INTERFACE I_CYLINDER_DA_TESTDEV2_4 EXTENDS I_CYLINDER_DA_GENERAL

METHOD M_OpenLockValves : BOOL
VAR_INPUT
  bOpenChA:        BOOL;
  bOpenChB:        BOOL;
END_VAR
END_METHOD

METHOD M_SetMaxPos : BOOL
VAR_INPUT
END_VAR
END_METHOD

METHOD M_SetZeroPos : BOOL
VAR_INPUT
END_VAR
END_METHOD

METHOD M_StopAndLock : BOOL
VAR_INPUT
END_VAR
END_METHOD

METHOD M_ToSetPos : BOOL
VAR_INPUT
  lrToSetPos:                 LREAL;
  /// Just need for prop valve
  eSpeedType:               E_SPEED_TYPE;
  rSpeed:                   REAL; 
END_VAR
END_METHOD

PROPERTY P_ActiveDirection : STRING
GET
END_GET
END_PROPERTY

PROPERTY P_DoubleActing : BOOL
GET
END_GET
END_PROPERTY

PROPERTY P_MaxPosVal : LREAL
GET
END_GET
END_PROPERTY

PROPERTY P_MinPosVal : LREAL
GET
END_GET
END_PROPERTY

PROPERTY P_Position : LREAL
GET
END_GET
END_PROPERTY

PROPERTY P_PositionAbs : LREAL
GET
END_GET
END_PROPERTY

PROPERTY P_PressureChA : REAL
GET
END_GET
END_PROPERTY

PROPERTY P_PressureChB : REAL
GET
END_GET
END_PROPERTY

PROPERTY P_SpeedInMmPerSecond : REAL
GET
END_GET
END_PROPERTY

PROPERTY P_SpeedInPercent : LREAL
GET
END_GET
END_PROPERTY

PROPERTY P_StrokeLength : REAL
GET
END_GET
END_PROPERTY

PROPERTY P_StrokeLengthInitialized : BOOL
GET
END_GET
SET
END_SET
END_PROPERTY

END_INTERFACE

(* stored: Version 1.1.0.1, ProductVersion 3.1.4024.12
   Itf I_CYLINDER_DA_TESTDEV2_4: Id {f16afa1c-8799-4f08-84e4-e0140353dd92}
   Method M_OpenLockValves: Id {2ca67dfe-0591-43a4-916c-384fb6af2657}
   Method M_SetMaxPos: Id {cea0ae47-e9bb-4f2e-bf7a-25e90d2d2955}
   Method M_SetZeroPos: Id {1ff466f2-f842-4159-9085-0bb5641ce510}
   Method M_StopAndLock: Id {74dc6512-611b-4bfe-84ef-8556535a1373}
   Method M_ToSetPos: Id {eded9da4-c374-40ff-b3c6-8b8ba669878d}
   Property P_ActiveDirection: Id {6203e25d-1d2e-4831-828b-3dd9d8c75aa4}
   Get Get: Id {7394b632-ea0c-48d3-9309-60833df95117}
   Property P_DoubleActing: Id {0b663a7c-7295-406b-b3e0-b046aa79acea}
   Get Get: Id {0442e461-205b-437a-97a8-3262d3e89e69}
   Property P_MaxPosVal: Id {75a29253-6f02-46db-8689-66b7709c9063}
   Get Get: Id {6d0277d3-aec1-4872-bee2-316417e4554c}
   Property P_MinPosVal: Id {3cce7030-0547-4c39-b29b-8a63b3db8061}
   Get Get: Id {818e9e8a-8ae0-49f1-8183-fb4253be33f4}
   Property P_Position: Id {aaf5d39b-950b-4fb4-9969-98f49b20be8b}
   Get Get: Id {bc82b54e-7ae4-4eab-8dd7-d6d38816469b}
   Property P_PositionAbs: Id {f5abc2d3-dc80-4dfb-9117-b9d4052ca3d4}
   Get Get: Id {22655590-92c2-4505-b7f6-7ba414aa1e6f}
   Property P_PressureChA: Id {2242dd50-d555-4854-9001-94346a7ea495}
   Get Get: Id {d7db13fa-f335-4081-9451-916fb814abc8}
   Property P_PressureChB: Id {07153e8d-795a-4709-a869-eb2aab084c16}
   Get Get: Id {b46329d2-2879-4ff8-8746-84792769ab21}
   Property P_SpeedInMmPerSecond: Id {301360ce-5962-4404-8936-dc0bc0f21f8a}
   Get Get: Id {9aeeef22-6037-4fbc-a70b-fc7a5fde3f85}
   Property P_SpeedInPercent: Id {a43fe268-c050-44b5-b0ec-529ff97cf970}
   Get Get: Id {1f066ded-0642-49b7-b50d-d9964f3cc570}
   Property P_StrokeLength: Id {55396f07-f6d7-4a30-97cd-1a505cf271ab}
   Get Get: Id {aecf620f-1882-4a23-ba5a-28bd14c0e87d}
   Property P_StrokeLengthInitialized: Id {d8f1c6b4-6813-4db6-b2e8-5b1f6496a57f}
   Get Get: Id {d8b23269-4ff5-4d93-b1b0-b56d480e0402}
   Set Set: Id {cdd192de-50b7-4b7f-be38-9356e9346f5a} *)
